# B&R Automation Studio project Genmot_Markalama_ (part 4)

#### GZ1Ax.c - Implementation code
```c
/*******************************************************************
 * COPYRIGHT -- Bernecker + Rainer
 ********************************************************************
 * PROGRAM: Basic
 * File: Basic.c
 * Author: Bernecker + Rainer
 * Created: December 01, 2009
 ********************************************************************
 * Implementation of Program Basic
 ********************************************************************/

#ifdef _DEFAULT_INCLUDES
#include <AsDefault.h>
#endif
#include <string.h>

/* defines of the state-constants */
#define STATE_WAIT              0
#define STATE_POWER_ON          1
#define STATE_HOME              2

#define STATE_READY             10
#define STATE_HALT              11
#define STATE_STOP              12
#define STATE_JOG_POSITIVE      13
#define STATE_JOG_NEGATIVE      14
#define STATE_MOVE_ABSOLUTE     15
#define STATE_MOVE_ADDITIVE     16
#define STATE_MOVE_VELOCITY     17

#define STATE_ERROR_AXIS        100
#define STATE_ERROR             101
#define STATE_ERROR_RESET       102
#define STATE_READ              103

_LOCAL REAL   data;

_INIT void GZ1Axis_init(void)
{

	/* get axis object */
	Axis1Obj = (UDINT)&GZ1_Axis;

	AxisStep = STATE_WAIT;  /* start step */

	GZ1Axis.Parameter.Velocity              = 10000;  /*velocity for movement*/
	GZ1Axis.Parameter.Acceleration          = 10000;  /*acceleration for movement*/
	GZ1Axis.Parameter.Deceleration          = 10000;  /*deceleration for movement*/
	GZ1Axis.Parameter.JogVelocity           = 5000;   /*velocity for jogging */

}

_CYCLIC void GZ1Axis_cyclic(void)
{
	if(GZ1Axis.Command.Power)
	{
		GZ1Axis.Speed.VelocityOverride			= 0.5;
	}

/***************************************************************
        Control Sequence
***************************************************************/

/* status information is read before the step sequencer to attain a shorter reaction time */
/************************ MC_READSTATUS *************************/
	MC_ReadStatus_0.Enable = !MC_ReadStatus_0.Error;
	MC_ReadStatus_0.Axis = Axis1Obj;
	MC_ReadStatus(&MC_ReadStatus_0);
	GZ1Axis.AxisState.Disabled             = MC_ReadStatus_0.Disabled;
	GZ1Axis.AxisState.StandStill           = MC_ReadStatus_0.StandStill;
	GZ1Axis.AxisState.Stopping             = MC_ReadStatus_0.Stopping;
	GZ1Axis.AxisState.Homing               = MC_ReadStatus_0.Homing;
	GZ1Axis.AxisState.DiscreteMotion       = MC_ReadStatus_0.DiscreteMotion;
	GZ1Axis.AxisState.ContinuousMotion     = MC_ReadStatus_0.ContinuousMotion;
	GZ1Axis.AxisState.SynchronizedMotion   = MC_ReadStatus_0.SynchronizedMotion;
	GZ1Axis.AxisState.ErrorStop            = MC_ReadStatus_0.Errorstop;

	/********************MC_BR_READDRIVESTATUS***********************/
	MC_BR_ReadDriveStatus_0.Enable = !MC_BR_ReadDriveStatus_0.Error;
	MC_BR_ReadDriveStatus_0.Axis = Axis1Obj;
	MC_BR_ReadDriveStatus_0.AdrDriveStatus = (UDINT)&(GZ1Axis.Status.DriveStatus);
	MC_BR_ReadDriveStatus(&MC_BR_ReadDriveStatus_0);

	/******************** MC_READACTUALPOSITION *********************/
	MC_ReadActualPosition_0.Enable = (!MC_ReadActualPosition_0.Error);
	MC_ReadActualPosition_0.Axis = Axis1Obj;
	MC_ReadActualPosition(&MC_ReadActualPosition_0);
	if(MC_ReadActualPosition_0.Valid == 1)
	{
		GZ1Axis.Status.ActPosition = MC_ReadActualPosition_0.Position;
	}

	/******************** MC_READACTUALVELOCITY *********************/
	MC_ReadActualVelocity_0.Enable = (!MC_ReadActualVelocity_0.Error);
	MC_ReadActualVelocity_0.Axis = Axis1Obj;
	MC_ReadActualVelocity(&MC_ReadActualVelocity_0);
	if(MC_ReadActualVelocity_0.Valid == 1)
	{
		GZ1Axis.Status.ActVelocity = MC_ReadActualVelocity_0.Velocity;
	}

	/*********************** MC SET OVERRIDE *********************/
	MC_SetOverride_0.Enable = (!MC_SetOverride_0.Error);
	MC_SetOverride_0.AccFactor = GZ1Axis.Speed.AccelerationOverride = 1.0;
	if ((GZ1Axis.Speed.VelocityOverride < 2.01) && (GZ1Axis.Speed.VelocityOverride > 0.0000001))
	{
		MC_SetOverride_0.VelFactor = GZ1Axis.Speed.VelocityOverride;
	}
	MC_SetOverride_0.Axis=Axis1Obj;
	MC_SetOverride(&MC_SetOverride_0);

	/************************ MC_READAXISERROR **********************/
	MC_ReadAxisError_0.Enable = !MC_ReadAxisError_0.Error;
	MC_ReadAxisError_0.Axis = Axis1Obj;
	MC_ReadAxisError_0.DataAddress = (UDINT)&(GZ1Axis.Status.ErrorText);
	MC_ReadAxisError_0.DataLength = sizeof(GZ1Axis.Status.ErrorText);
	strcpy((void*)&MC_ReadAxisError_0.DataObjectName,"acp10etxen");
	MC_ReadAxisError(&MC_ReadAxisError_0);

	/* central monitoring of stop command attains a shorter reaction time in case of emergency stop */
	/******************CHECK for STOP COMMAND************************/
	if (GZ1Axis.Command.Stop == 1)
	{
		if ((AxisStep >= STATE_READY) && (AxisStep < STATE_ERROR))
		{
			/* reset all FB execute inputs we use */
			MC_Home_0.Execute = 0;
			MC_Stop_0.Execute = 0;
			MC_MoveAbsolute_0.Execute = 0;
			MC_MoveAdditive_0.Execute = 0;
			MC_MoveVelocity_0.Execute = 0;
			MC_ReadAxisError_0.Acknowledge = 0;
			MC_Reset_0.Execute = 0;

			/* reset user commands */
			GZ1Axis.Command.Stop = 0;
			GZ1Axis.Command.Home = 0;
			GZ1Axis.Command.MoveJogPos = 0;
			GZ1Axis.Command.MoveJogNeg = 0;
			GZ1Axis.Command.MoveVelocity = 0;
			GZ1Axis.Command.MoveAbsolute = 0;
			GZ1Axis.Command.MoveAdditive = 0;
			AxisStep = STATE_STOP;
		}
	}

	/**************** CHECK FOR GENERAL AXIS ERROR ******************/
	if ((MC_ReadAxisError_0.AxisErrorID != 0) && (MC_ReadAxisError_0.Valid == 1))
	{
		AxisStep = STATE_ERROR_AXIS;
	}
		/***************** CHECK IF POWER SHOULD BE OFF *******************/
	else if ((GZ1Axis.Command.Power == 0) && (MC_ReadAxisError_0.Valid == 1))
	{
		if ((MC_ReadStatus_0.Errorstop == 1) && (MC_ReadStatus_0.Valid == 1))
		{
			AxisStep = STATE_ERROR_RESET;
		}
		else
		{
			AxisStep = STATE_WAIT;
		}
	}

	switch(AxisStep)
	{
		/******************** WAIT *************************/
		case STATE_WAIT:  /* STATE: Wait */
			if (GZ1Axis.Command.Power == 1)
			{
				AxisStep = STATE_POWER_ON;
			}
			else
			{
				MC_Power_0.Enable = 0;

			}

			/* reset all FB execute inputs we use */
			MC_Home_0.Execute = 0;
			MC_Stop_0.Execute = 0;
			MC_MoveAbsolute_0.Execute = 0;
			MC_MoveAdditive_0.Execute = 0;
			MC_MoveVelocity_0.Execute = 0;
			MC_ReadAxisError_0.Acknowledge = 0;
			MC_Reset_0.Execute = 0;

			/* reset user commands */
			GZ1Axis.Command.Stop = 0;
			GZ1Axis.Command.Home = 0;
			GZ1Axis.Command.MoveJogPos = 0;
			GZ1Axis.Command.MoveJogNeg = 0;
			GZ1Axis.Command.MoveVelocity = 0;
			GZ1Axis.Command.MoveAbsolute = 0;
			GZ1Axis.Command.MoveAdditive = 0;

			GZ1Axis.Status.ErrorID = 0;
			break;

		/******************** POWER ON **********************/
		case STATE_POWER_ON:  /* STATE: Power on */
			MC_Power_0.Enable = 1;
			if (MC_Power_0.Status == 1)
			{
				if (!GZ1HomeOk & Parametreler_0.Z_HomeStart)
				{
					GZ1Axis.Command.Home = 1;
				}
			    AxisStep = STATE_READY;
			}
			/* if a power error occured go to error state */
			if (MC_Power_0.Error == 1)
			{
				GZ1Axis.Status.ErrorID = MC_Power_0.ErrorID;
				AxisStep = STATE_ERROR;
			}
			break;

		/******************** READY **********************/
		case STATE_READY:  /* STATE: Waiting for commands */
			if (GZ1Axis.Command.Home == 1)
			{
				GZ1Axis.Command.Home = 0;
				AxisStep = STATE_HOME;
			}
			else if (GZ1Axis.Command.Stop == 1)
			{
				AxisStep = STATE_STOP;
			}
			else if (GZ1Axis.Command.MoveJogPos == 1)
			{
				AxisStep = STATE_JOG_POSITIVE;
			}
			else if (GZ1Axis.Command.MoveJogNeg == 1)
			{
				AxisStep = STATE_JOG_NEGATIVE;
			}
			else if (GZ1Axis.Command.MoveAbsolute == 1)
			{
				GZ1Axis.Command.MoveAbsolute = 0;
				AxisStep = STATE_MOVE_ABSOLUTE;
			}
			else if (GZ1Axis.Command.MoveAdditive == 1)
			{
				GZ1Axis.Command.MoveAdditive = 0;
				AxisStep = STATE_MOVE_ADDITIVE;
			}
			else if (GZ1Axis.Command.MoveVelocity == 1)
			{
				GZ1Axis.Command.MoveVelocity = 0;
				AxisStep = STATE_MOVE_VELOCITY;
			}
			else if (GZ1Axis.Command.Halt == 1)
			{
				GZ1Axis.Command.Halt = 0;
				AxisStep = STATE_HALT;
			}
			break;

		/******************** HOME **********************/
		case STATE_HOME:  /* STATE: start homing process */
			MC_Home_0.Position = GZ1Axis.Parameter.HomePosition;
			MC_Home_0.HomingMode = GZ1Axis.Parameter.HomeMode;
			MC_Home_0.Execute = 1;
			if (MC_Home_0.Done == 1)
			{

				MC_Home_0.Execute = 0;
				AxisStep = STATE_READ;
			}
			/* if a homing error occured go to error state */
			if (MC_Home_0.Error == 1)
			{
				MC_Home_0.Execute = 0;
				GZ1Axis.Status.ErrorID = MC_Home_0.ErrorID;
				AxisStep = STATE_ERROR;
			}
			break;

		/************************HALT MOVEMENT**************************/
		case STATE_HALT:  /* STATE: Stop the active movement */
			MC_Halt_0.Deceleration = GZ1Axis.Parameter.Deceleration;
			MC_Halt_0.Execute = 1;
			if (MC_Halt_0.Done == 1)
			{
				MC_Halt_0.Execute = 0;
				AxisStep = STATE_READY;
			}
			/*check if error occured */
			if (MC_Halt_0.Error == 1)
			{
				MC_Halt_0.Execute = 0;
				GZ1Axis.Status.ErrorID = MC_Halt_0.ErrorID;
				AxisStep = STATE_ERROR;
			}
			break;

		/*********************** STOP MOVEMENT *************************/
		case STATE_STOP: /* STATE: Stop movement as long as command is set */
			MC_Stop_0.Deceleration = GZ1Axis.Parameter.Deceleration;
			MC_Stop_0.Execute = 1;
			/* if axis is stopped go to ready state */
			if ((MC_Stop_0.Done == 1) && (GZ1Axis.Command.Stop == 0))
			{
				MC_Stop_0.Execute = 0;
				AxisStep = STATE_READY;
			}
			/* check if error occured */
			if (MC_Stop_0.Error == 1)
			{
				GZ1Axis.Status.ErrorID = MC_Stop_0.ErrorID;
				MC_Stop_0.Execute = 0;
				AxisStep = STATE_ERROR;
			}
			break;

		/******************** START JOG MOVEMENT POSITVE **********************/
		case STATE_JOG_POSITIVE:  /* STATE: Start jog movement in positive direction */
			MC_MoveVelocity_0.Velocity      = GZ1Axis.Parameter.JogVelocity;
			MC_MoveVelocity_0.Acceleration  = GZ1Axis.Parameter.Acceleration;
			MC_MoveVelocity_0.Deceleration  = GZ1Axis.Parameter.Deceleration;
			MC_MoveVelocity_0.Direction     = mcPOSITIVE_DIR;
			MC_MoveVelocity_0.Execute = 1;
			/* check if jog movement should be stopped */
			if (GZ1Axis.Command.MoveJogPos == 0)
			{
				MC_MoveVelocity_0.Execute = 0;
				AxisStep = STATE_HALT;
			}
			/* check if error occured */
			if (MC_MoveVelocity_0.Error == 1)
			{
				GZ1Axis.Status.ErrorID = MC_MoveVelocity_0.ErrorID;
				MC_MoveVelocity_0.Execute = 0;
				AxisStep = STATE_ERROR;
			}
			break;

		/******************** START JOG MOVEMENT NEGATIVE **********************/
		case STATE_JOG_NEGATIVE:  /* STATE: Start jog movement in negative direction */
			MC_MoveVelocity_0.Velocity      = GZ1Axis.Parameter.JogVelocity;
			MC_MoveVelocity_0.Acceleration  = GZ1Axis.Parameter.Acceleration;
			MC_MoveVelocity_0.Deceleration  = GZ1Axis.Parameter.Deceleration;
			MC_MoveVelocity_0.Direction     = mcNEGATIVE_DIR;
			MC_MoveVelocity_0.Execute = 1;
			/* check if jog movement should be stopped */
			if (GZ1Axis.Command.MoveJogNeg == 0)
			{
				MC_MoveVelocity_0.Execute = 0;
				AxisStep = STATE_HALT;
			}
			/* check if error occured */
			if (MC_MoveVelocity_0.Error == 1)
			{
				GZ1Axis.Status.ErrorID = MC_MoveVelocity_0.ErrorID;
				MC_MoveVelocity_0.Execute = 0;
				AxisStep = STATE_ERROR;
			}
			break;

		/******************** START ABSOLUTE MOVEMENT **********************/
		case STATE_MOVE_ABSOLUTE:  /* STATE: Start absolute movement */
			MC_MoveAbsolute_0.Position      = GZ1Axis.Parameter.Position;
			MC_MoveAbsolute_0.Velocity      = GZ1Axis.Parameter.Velocity;
			MC_MoveAbsolute_0.Acceleration  = GZ1Axis.Parameter.Acceleration;
			MC_MoveAbsolute_0.Deceleration  = GZ1Axis.Parameter.Deceleration;
			MC_MoveAbsolute_0.Direction     = GZ1Axis.Parameter.Direction;
			MC_MoveAbsolute_0.Execute = 1;
			/* check if commanded position is reached */
			if (GZ1Axis.Command.Halt == 1)
			{
				GZ1Axis.Command.Halt = 0;
				MC_MoveAbsolute_0.Execute = 0;
				AxisStep = STATE_HALT;
			}
			else if (MC_MoveAbsolute_0.Done == 1)
			{
				MC_MoveAbsolute_0.Execute = 0;
				AxisStep = STATE_READY;
			}
			/* check if error occured */
			if (MC_MoveAbsolute_0.Error == 1)
			{
				GZ1Axis.Status.ErrorID = MC_MoveAbsolute_0.ErrorID;
				MC_MoveAbsolute_0.Execute = 0;
				AxisStep = STATE_ERROR;
			}
			break;

		/******************** START ADDITIVE MOVEMENT **********************/
		case STATE_MOVE_ADDITIVE:  /* STATE: Start additive movement */
			MC_MoveAdditive_0.Distance      = GZ1Axis.Parameter.Distance;
			MC_MoveAdditive_0.Velocity      = GZ1Axis.Parameter.Velocity;
			MC_MoveAdditive_0.Acceleration  = GZ1Axis.Parameter.Acceleration;
			MC_MoveAdditive_0.Deceleration  = GZ1Axis.Parameter.Deceleration;
			MC_MoveAdditive_0.Execute = 1;
			/* check if commanded distance is reached */
			if (GZ1Axis.Command.Halt == 1)
			{
				GZ1Axis.Command.Halt = 0;
				MC_MoveAdditive_0.Execute = 0;
				AxisStep = STATE_HALT;
			}
			else if (MC_MoveAdditive_0.Done == 1)
			{
				MC_MoveAdditive_0.Execute = 0;
				AxisStep = STATE_READY;
			}
			/* check if error occured */
			if (MC_MoveAdditive_0.Error == 1)
			{
				GZ1Axis.Status.ErrorID = MC_MoveAdditive_0.ErrorID;
				MC_MoveAdditive_0.Execute = 0;
				AxisStep = STATE_ERROR;
			}
			break;

		/******************** START VELOCITY MOVEMENT **********************/
		case STATE_MOVE_VELOCITY:  /* STATE: Start velocity movement */
			MC_MoveVelocity_0.Velocity      = GZ1Axis.Parameter.Velocity;
			MC_MoveVelocity_0.Acceleration  = GZ1Axis.Parameter.Acceleration;
			MC_MoveVelocity_0.Deceleration  = GZ1Axis.Parameter.Deceleration;
			MC_MoveVelocity_0.Direction     = GZ1Axis.Parameter.Direction;
			MC_MoveVelocity_0.Execute = 1;
			/* check if commanded velocity is reached */
			if (GZ1Axis.Command.Halt == 1)
			{
				GZ1Axis.Command.Halt = 0;
				MC_MoveVelocity_0.Execute = 0;
				AxisStep = STATE_HALT;
			}
			else if (MC_MoveVelocity_0.InVelocity == 1)
			{
				MC_MoveVelocity_0.Execute = 0;
				AxisStep = STATE_READY;
			}
			/* check if error occured */
			if (MC_MoveVelocity_0.Error == 1)
			{
				GZ1Axis.Status.ErrorID = MC_MoveVelocity_0.ErrorID;
				MC_MoveVelocity_0.Execute = 0;
				AxisStep = STATE_ERROR;
			}
			break;

		/******************** FB-ERROR OCCURED *************************/
		case STATE_ERROR:  /* STATE: Error */
			/* check if FB indicates an axis error */
			if (MC_ReadAxisError_0.AxisErrorCount != 0)
			{
				AxisStep = STATE_ERROR_AXIS;
			}
			else
			{
				if (GZ1Axis.Command.ErrorAcknowledge == 1)
				{
					GZ1Axis.Command.ErrorAcknowledge = 0;
					GZ1Axis.Status.ErrorID = 0;
					/* reset axis if it is in axis state ErrorStop */
					if ((MC_ReadStatus_0.Errorstop == 1) && (MC_ReadStatus_0.Valid == 1))
					{
						AxisStep = STATE_ERROR_RESET;
					}
					else
					{
						AxisStep = STATE_WAIT;
					}
				}
			}
			break;

		/******************** AXIS-ERROR OCCURED *************************/
		case STATE_ERROR_AXIS:  /* STATE: Axis Error */
			if (MC_ReadAxisError_0.Valid == 1)
			{
				if (MC_ReadAxisError_0.AxisErrorID != 0)
				{
					GZ1Axis.Status.ErrorID = MC_ReadAxisError_0.AxisErrorID;
				}
				MC_ReadAxisError_0.Acknowledge = 0;
				if (GZ1Axis.Command.ErrorAcknowledge == 1)
				{
					GZ1Axis.Command.ErrorAcknowledge = 0;
					/* acknowledge axis error */
					if (MC_ReadAxisError_0.AxisErrorID != 0)
					{
						MC_ReadAxisError_0.Acknowledge = 1;
					}
				}
				if (MC_ReadAxisError_0.AxisErrorCount == 0)
				{
					GZ1Axis.Status.ErrorID = 0;
					/* reset axis if it is in axis state ErrorStop */
					if ((MC_ReadStatus_0.Errorstop == 1) && (MC_ReadStatus_0.Valid == 1))
					{
						AxisStep = STATE_ERROR_RESET;
					}
					else
					{
						AxisStep = STATE_WAIT;
					}
				}
			}
			break;

		/******************** RESET DONE *************************/
		case STATE_ERROR_RESET:  /* STATE: Wait for reset done */
			MC_Reset_0.Execute = 1;
			/* reset MC_Power.Enable if this FB is in Error*/
			if(MC_Power_0.Error == 1)
			{
				MC_Power_0.Enable = 0;
			}
			if(MC_Reset_0.Done == 1)
			{
				MC_Reset_0.Execute = 0;
				AxisStep = STATE_WAIT;
			}
			else if (MC_Reset_0.Error == 1)
			{
				MC_Reset_0.Execute = 0;
				AxisStep = STATE_ERROR;
			}
			break;

		/******************** SEQUENCE END *************************/

		/**********************STATE_READ************************/
		case STATE_READ:
			MC_BR_CyclicRead_0.Enable=1;
			MC_BR_CyclicRead_0.ParID = 277;
			MC_BR_CyclicRead_0.DataAddress = (UDINT)&data;
			MC_BR_CyclicRead_0.DataType =ncPAR_TYP_REAL;

			if (MC_BR_CyclicRead_0.Valid)
			{
				AxisStep = STATE_READY;
			}
			else if (MC_BR_CyclicRead_0.Error)
			{

				GZ1Axis.Status.ErrorID = MC_BR_CyclicRead_0.ErrorID;
				/*Reset Enable before going to STATE_ERROR*/
				MC_BR_CyclicRead_0.Enable=0;
				AxisStep = STATE_ERROR;
			}
			break;  /*end read*/

	}

/***************************************************************
        Function Block Calls
***************************************************************/

/************************** MC_POWER ****************************/
	MC_Power_0.Axis = Axis1Obj;  /* pointer to axis */
	MC_Power(&MC_Power_0);

	/************************** MC_HOME *****************************/
	MC_Home_0.Axis = Axis1Obj;
	MC_Home(&MC_Home_0);

	/********************** MC_MOVEABSOLUTE *************************/
	MC_MoveAbsolute_0.Axis = Axis1Obj;
	MC_MoveAbsolute(&MC_MoveAbsolute_0);

	/********************** MC_MOVEADDITIVE *************************/
	MC_MoveAdditive_0.Axis = Axis1Obj;
	MC_MoveAdditive(&MC_MoveAdditive_0);

	/********************** MC_MOVEVELOCITY *************************/
	MC_MoveVelocity_0.Axis = Axis1Obj;
	MC_MoveVelocity(&MC_MoveVelocity_0);

	/************************** MC_STOP *****************************/
	MC_Stop_0.Axis = Axis1Obj;
	MC_Stop(&MC_Stop_0);

	/**************************MC_HALT*******************************/
	MC_Halt_0.Axis = Axis1Obj;
	MC_Halt(&MC_Halt_0);

	/************************** MC_RESET ****************************/
	MC_Reset_0.Axis = Axis1Obj;
	MC_Reset(&MC_Reset_0);

	MC_BR_CyclicRead_0.Axis = Axis1Obj;
	MC_BR_CyclicRead(&MC_BR_CyclicRead_0);

}
```

#### GZ1Ax.var - Local variables
```iecst
(********************************************************************
 * COPYRIGHT --
 ********************************************************************
 * Program: Reg2Ax
 * File: Reg2Ax.var
 * Author: Coder
 * Created: June 20, 2013
 ********************************************************************
 * Local variables of program Reg2Ax
 ********************************************************************)
VAR
	Axis1Obj : UDINT; (*axis reference*)
	Axis2Obj : UDINT; (*axis reference*)
	AxisStep : USINT; (*current step in the step sequence*)
	AutData : MC_AUTDATA_TYP := (0); (*configuration of the automat*)
	MC_Power_0 : MC_Power; (*Function Block*)
	MC_Home_0 : MC_Home; (*Function Block*)
	MC_Stop_0 : MC_Stop; (*Function Block*)
	MC_MoveVelocity_0 : MC_MoveVelocity; (*Function Block*)
	MC_MoveAbsolute_0 : MC_MoveAbsolute; (*Function Block*)
	MC_MoveAdditive_0 : MC_MoveAdditive; (*Function Block*)
	MC_BR_InitAutData_0 : MC_BR_InitAutData; (*Function Block*)
	MC_BR_AutControl_0 : MC_BR_AutControl; (*Function Block*)
	MC_ReadAxisError_0 : MC_ReadAxisError; (*Function Block*)
	MC_Reset_0 : MC_Reset; (*Function Block*)
	MC_ReadStatus_0 : MC_ReadStatus; (*Function Block*)
	MC_ReadActualPosition_0 : MC_ReadActualPosition; (*Function Block*)
	MC_ReadActualVelocity_0 : MC_ReadActualVelocity; (*Function Block*)
	MC_BR_ReadDriveStatus_0 : MC_BR_ReadDriveStatus; (*Function Block*)
	MC_Halt_0 : MC_Halt; (*Function Block*)
	MC_BR_DownloadCamProfileObj_0 : MC_BR_DownloadCamProfileObj;
	SlaveFactor : REAL;
	MC_BR_Phasing_0 : MC_BR_Phasing;
	ShiftFactor : REAL;
	MC_GearInPos_0 : MC_GearInPos;
	MC_GearOut_0 : MC_GearOut;
	MC_SetOverride_0 : MC_SetOverride;
	MC_BR_CyclicRead_0 : MC_BR_CyclicRead;
END_VAR
```

### Program Logical/RC1AxisControl (ANSIC)

#### GC1Ax.c - Implementation code
```c
/*******************************************************************
 * COPYRIGHT -- Bernecker + Rainer
 ********************************************************************
 * PROGRAM: Basic
 * File: Basic.c
 * Author: Bernecker + Rainer
 * Created: December 01, 2009
 ********************************************************************
 * Implementation of Program Basic
 ********************************************************************/

#ifdef _DEFAULT_INCLUDES
#include <AsDefault.h>
#endif
#include <string.h>

/* defines of the state-constants */
#define STATE_WAIT              0
#define STATE_POWER_ON          1
#define STATE_HOME              2

#define STATE_READY             10
#define STATE_HALT              11
#define STATE_STOP              12
#define STATE_JOG_POSITIVE      13
#define STATE_JOG_NEGATIVE      14
#define STATE_MOVE_ABSOLUTE     15
#define STATE_MOVE_ADDITIVE     16
#define STATE_MOVE_VELOCITY     17

#define STATE_ERROR_AXIS        100
#define STATE_ERROR             101
#define STATE_ERROR_RESET       102
#define STATE_READ              103

_LOCAL REAL   data;

_INIT void GC1Axis_init(void)
{

	/* get axis object */
	Axis1Obj = (UDINT)&GC1_Axis;

	AxisStep = STATE_WAIT;  /* start step */

	GC1Axis.Parameter.Velocity              = 2000;  /*velocity for movement*/
	GC1Axis.Parameter.Acceleration          = 10000;  /*acceleration for movement*/
	GC1Axis.Parameter.Deceleration          = 10000;  /*deceleration for movement*/
	GC1Axis.Parameter.JogVelocity           = 2000;   /*velocity for jogging */

}

_CYCLIC void GC1Axis_cyclic(void)
{
	if(GC1Axis.Command.Power)
	{
		GC1Axis.Speed.VelocityOverride			= 0.5;
	}

/***************************************************************
        Control Sequence
***************************************************************/

/* status information is read before the step sequencer to attain a shorter reaction time */
/************************ MC_READSTATUS *************************/
	MC_ReadStatus_0.Enable = !MC_ReadStatus_0.Error;
	MC_ReadStatus_0.Axis = Axis1Obj;
	MC_ReadStatus(&MC_ReadStatus_0);
	GC1Axis.AxisState.Disabled             = MC_ReadStatus_0.Disabled;
	GC1Axis.AxisState.StandStill           = MC_ReadStatus_0.StandStill;
	GC1Axis.AxisState.Stopping             = MC_ReadStatus_0.Stopping;
	GC1Axis.AxisState.Homing               = MC_ReadStatus_0.Homing;
	GC1Axis.AxisState.DiscreteMotion       = MC_ReadStatus_0.DiscreteMotion;
	GC1Axis.AxisState.ContinuousMotion     = MC_ReadStatus_0.ContinuousMotion;
	GC1Axis.AxisState.SynchronizedMotion   = MC_ReadStatus_0.SynchronizedMotion;
	GC1Axis.AxisState.ErrorStop            = MC_ReadStatus_0.Errorstop;

	/********************MC_BR_READDRIVESTATUS***********************/
	MC_BR_ReadDriveStatus_0.Enable = !MC_BR_ReadDriveStatus_0.Error;
	MC_BR_ReadDriveStatus_0.Axis = Axis1Obj;
	MC_BR_ReadDriveStatus_0.AdrDriveStatus = (UDINT)&(GC1Axis.Status.DriveStatus);
	MC_BR_ReadDriveStatus(&MC_BR_ReadDriveStatus_0);

	/******************** MC_READACTUALPOSITION *********************/
	MC_ReadActualPosition_0.Enable = (!MC_ReadActualPosition_0.Error);
	MC_ReadActualPosition_0.Axis = Axis1Obj;
	MC_ReadActualPosition(&MC_ReadActualPosition_0);
	if(MC_ReadActualPosition_0.Valid == 1)
	{
		GC1Axis.Status.ActPosition = MC_ReadActualPosition_0.Position;
	}

	/******************** MC_READACTUALVELOCITY *********************/
	MC_ReadActualVelocity_0.Enable = (!MC_ReadActualVelocity_0.Error);
	MC_ReadActualVelocity_0.Axis = Axis1Obj;
	MC_ReadActualVelocity(&MC_ReadActualVelocity_0);
	if(MC_ReadActualVelocity_0.Valid == 1)
	{
		GC1Axis.Status.ActVelocity = MC_ReadActualVelocity_0.Velocity;
	}

	/*********************** MC SET OVERRIDE *********************/
	MC_SetOverride_0.Enable = (!MC_SetOverride_0.Error);
	MC_SetOverride_0.AccFactor = GC1Axis.Speed.AccelerationOverride = 1.0;
	if ((GC1Axis.Speed.VelocityOverride < 2.01) && (GC1Axis.Speed.VelocityOverride > 0.0000001))
	{
		MC_SetOverride_0.VelFactor = GC1Axis.Speed.VelocityOverride;
	}
	MC_SetOverride_0.Axis=Axis1Obj;
	MC_SetOverride(&MC_SetOverride_0);

	/************************ MC_READAXISERROR **********************/
	MC_ReadAxisError_0.Enable = !MC_ReadAxisError_0.Error;
	MC_ReadAxisError_0.Axis = Axis1Obj;
	MC_ReadAxisError_0.DataAddress = (UDINT)&(GC1Axis.Status.ErrorText);
	MC_ReadAxisError_0.DataLength = sizeof(GC1Axis.Status.ErrorText);
	strcpy((void*)&MC_ReadAxisError_0.DataObjectName,"acp10etxen");
	MC_ReadAxisError(&MC_ReadAxisError_0);

	/* central monitoring of stop command attains a shorter reaction time in case of emergency stop */
	/******************CHECK for STOP COMMAND************************/
	if (GC1Axis.Command.Stop == 1)
	{
		if ((AxisStep >= STATE_READY) && (AxisStep < STATE_ERROR))
		{
			/* reset all FB execute inputs we use */
			MC_Home_0.Execute = 0;
			MC_Stop_0.Execute = 0;
			MC_MoveAbsolute_0.Execute = 0;
			MC_MoveAdditive_0.Execute = 0;
			MC_MoveVelocity_0.Execute = 0;
			MC_ReadAxisError_0.Acknowledge = 0;
			MC_Reset_0.Execute = 0;

			/* reset user commands */
			GC1Axis.Command.Stop = 0;
			GC1Axis.Command.Home = 0;
			GC1Axis.Command.MoveJogPos = 0;
			GC1Axis.Command.MoveJogNeg = 0;
			GC1Axis.Command.MoveVelocity = 0;
			GC1Axis.Command.MoveAbsolute = 0;
			GC1Axis.Command.MoveAdditive = 0;
			AxisStep = STATE_STOP;
		}
	}

	/**************** CHECK FOR GENERAL AXIS ERROR ******************/
	if ((MC_ReadAxisError_0.AxisErrorID != 0) && (MC_ReadAxisError_0.Valid == 1))
	{
		AxisStep = STATE_ERROR_AXIS;
	}
		/***************** CHECK IF POWER SHOULD BE OFF *******************/
	else if ((GC1Axis.Command.Power == 0) && (MC_ReadAxisError_0.Valid == 1))
	{
		if ((MC_ReadStatus_0.Errorstop == 1) && (MC_ReadStatus_0.Valid == 1))
		{
			AxisStep = STATE_ERROR_RESET;
		}
		else
		{
			AxisStep = STATE_WAIT;
		}
	}

	switch(AxisStep)
	{
		/******************** WAIT *************************/
		case STATE_WAIT:  /* STATE: Wait */
			if (GC1Axis.Command.Power == 1)
			{
				AxisStep = STATE_POWER_ON;
			}
			else
			{
				MC_Power_0.Enable = 0;

			}

			/* reset all FB execute inputs we use */
			MC_Home_0.Execute = 0;
			MC_Stop_0.Execute = 0;
			MC_MoveAbsolute_0.Execute = 0;
			MC_MoveAdditive_0.Execute = 0;
			MC_MoveVelocity_0.Execute = 0;
			MC_ReadAxisError_0.Acknowledge = 0;
			MC_Reset_0.Execute = 0;

			/* reset user commands */
			GC1Axis.Command.Stop = 0;
			GC1Axis.Command.Home = 0;
			GC1Axis.Command.MoveJogPos = 0;
			GC1Axis.Command.MoveJogNeg = 0;
			GC1Axis.Command.MoveVelocity = 0;
			GC1Axis.Command.MoveAbsolute = 0;
			GC1Axis.Command.MoveAdditive = 0;

			GC1Axis.Status.ErrorID = 0;
			break;

		/******************** POWER ON **********************/
		case STATE_POWER_ON:  /* STATE: Power on */
			MC_Power_0.Enable = 1;
			if (MC_Power_0.Status == 1)
			{
				if (Parametreler_0.GC1_HomeStart)
				{
					GC1Axis.Command.Home = 1;
				}
			    AxisStep = STATE_READY;
			}
			/* if a power error occured go to error state */
			if (MC_Power_0.Error == 1)
			{
				GC1Axis.Status.ErrorID = MC_Power_0.ErrorID;
				AxisStep = STATE_ERROR;
			}
			break;

		/******************** READY **********************/
		case STATE_READY:  /* STATE: Waiting for commands */
			if (GC1Axis.Command.Home == 1)
			{
				GC1Axis.Command.Home = 0;
				AxisStep = STATE_HOME;
			}
			else if (GC1Axis.Command.Stop == 1)
			{
				AxisStep = STATE_STOP;
			}
			else if (GC1Axis.Command.MoveJogPos == 1)
			{
				AxisStep = STATE_JOG_POSITIVE;
			}
			else if (GC1Axis.Command.MoveJogNeg == 1)
			{
				AxisStep = STATE_JOG_NEGATIVE;
			}
			else if (GC1Axis.Command.MoveAbsolute == 1)
			{
				GC1Axis.Command.MoveAbsolute = 0;
				AxisStep = STATE_MOVE_ABSOLUTE;
			}
			else if (GC1Axis.Command.MoveAdditive == 1)
			{
				GC1Axis.Command.MoveAdditive = 0;
				AxisStep = STATE_MOVE_ADDITIVE;
			}
			else if (GC1Axis.Command.MoveVelocity == 1)
			{
				GC1Axis.Command.MoveVelocity = 0;
				AxisStep = STATE_MOVE_VELOCITY;
			}
			else if (GC1Axis.Command.Halt == 1)
			{
				GC1Axis.Command.Halt = 0;
				AxisStep = STATE_HALT;
			}
			break;

		/******************** HOME **********************/
		case STATE_HOME:  /* STATE: start homing process */
			if (!GC2Axis.AxisState.SynchronizedMotion)
			{
				MC_Home_0.Position = GC1Axis.Parameter.HomePosition;
				MC_Home_0.HomingMode = GC1Axis.Parameter.HomeMode;
				MC_Home_0.Execute = 1;
				if (MC_Home_0.Done == 1 )
				{
					//

					MC_Home_0.Execute = 0;
					AxisStep = STATE_READ;
				}
				/* if a homing error occured go to error state */
				if (MC_Home_0.Error == 1)
				{
					MC_Home_0.Execute = 0;
					GC1Axis.Status.ErrorID = MC_Home_0.ErrorID;
					AxisStep = STATE_ERROR;
				}
			}
			else
			{
				AxisStep = STATE_READ;
				GC2Axis.Command.GearOut = 1;
				GC2Axis.Command.GearInPos = 0;

			}
			break;

		/************************HALT MOVEMENT**************************/
		case STATE_HALT:  /* STATE: Stop the active movement */
			MC_Halt_0.Deceleration = GC1Axis.Parameter.Deceleration;
			MC_Halt_0.Execute = 1;
			if (MC_Halt_0.Done == 1)
			{
				MC_Halt_0.Execute = 0;
				AxisStep = STATE_READY;
			}
			/*check if error occured */
			if (MC_Halt_0.Error == 1)
			{
				MC_Halt_0.Execute = 0;
				GC1Axis.Status.ErrorID = MC_Halt_0.ErrorID;
				AxisStep = STATE_ERROR;
			}
			break;

		/*********************** STOP MOVEMENT *************************/
		case STATE_STOP: /* STATE: Stop movement as long as command is set */
			MC_Stop_0.Deceleration = GC1Axis.Parameter.Deceleration;
			MC_Stop_0.Execute = 1;
			/* if axis is stopped go to ready state */
			if ((MC_Stop_0.Done == 1) && (GC1Axis.Command.Stop == 0))
			{
				MC_Stop_0.Execute = 0;
				AxisStep = STATE_READY;
			}
			/* check if error occured */
			if (MC_Stop_0.Error == 1)
			{
				GC1Axis.Status.ErrorID = MC_Stop_0.ErrorID;
				MC_Stop_0.Execute = 0;
				AxisStep = STATE_ERROR;
			}
			break;

		/******************** START JOG MOVEMENT POSITVE **********************/
		case STATE_JOG_POSITIVE:  /* STATE: Start jog movement in positive direction */
			MC_MoveVelocity_0.Velocity      = GC1Axis.Parameter.JogVelocity;
			MC_MoveVelocity_0.Acceleration  = GC1Axis.Parameter.Acceleration;
			MC_MoveVelocity_0.Deceleration  = GC1Axis.Parameter.Deceleration;
			MC_MoveVelocity_0.Direction     = mcPOSITIVE_DIR;
			MC_MoveVelocity_0.Execute = 1;
			/* check if jog movement should be stopped */
			if (GC1Axis.Command.MoveJogPos == 0)
			{
				MC_MoveVelocity_0.Execute = 0;
				AxisStep = STATE_HALT;
			}
			/* check if error occured */
			if (MC_MoveVelocity_0.Error == 1)
			{
				GC1Axis.Status.ErrorID = MC_MoveVelocity_0.ErrorID;
				MC_MoveVelocity_0.Execute = 0;
				AxisStep = STATE_ERROR;
			}
			break;

		/******************** START JOG MOVEMENT NEGATIVE **********************/
		case STATE_JOG_NEGATIVE:  /* STATE: Start jog movement in negative direction */
			MC_MoveVelocity_0.Velocity      = GC1Axis.Parameter.JogVelocity;
			MC_MoveVelocity_0.Acceleration  = GC1Axis.Parameter.Acceleration;
			MC_MoveVelocity_0.Deceleration  = GC1Axis.Parameter.Deceleration;
			MC_MoveVelocity_0.Direction     = mcNEGATIVE_DIR;
			MC_MoveVelocity_0.Execute = 1;
			/* check if jog movement should be stopped */
			if (GC1Axis.Command.MoveJogNeg == 0)
			{
				MC_MoveVelocity_0.Execute = 0;
				AxisStep = STATE_HALT;
			}
			/* check if error occured */
			if (MC_MoveVelocity_0.Error == 1)
			{
				GC1Axis.Status.ErrorID = MC_MoveVelocity_0.ErrorID;
				MC_MoveVelocity_0.Execute = 0;
				AxisStep = STATE_ERROR;
			}
			break;

		/******************** START ABSOLUTE MOVEMENT **********************/
		case STATE_MOVE_ABSOLUTE:  /* STATE: Start absolute movement */
			MC_MoveAbsolute_0.Position      = GC1Axis.Parameter.Position;
			MC_MoveAbsolute_0.Velocity      = GC1Axis.Parameter.Velocity;
			MC_MoveAbsolute_0.Acceleration  = GC1Axis.Parameter.Acceleration;
			MC_MoveAbsolute_0.Deceleration  = GC1Axis.Parameter.Deceleration;
			MC_MoveAbsolute_0.Direction     = GC1Axis.Parameter.Direction;
			MC_MoveAbsolute_0.Execute = 1;
			/* check if commanded position is reached */
			if (GC1Axis.Command.Halt == 1)
			{
				GC1Axis.Command.Halt = 0;
				MC_MoveAbsolute_0.Execute = 0;
				AxisStep = STATE_HALT;
			}
			else if (MC_MoveAbsolute_0.Done == 1)
			{
				MC_MoveAbsolute_0.Execute = 0;
				AxisStep = STATE_READY;
			}
			/* check if error occured */
			if (MC_MoveAbsolute_0.Error == 1)
			{
				GC1Axis.Status.ErrorID = MC_MoveAbsolute_0.ErrorID;
				MC_MoveAbsolute_0.Execute = 0;
				AxisStep = STATE_ERROR;
			}
			break;

		/******************** START ADDITIVE MOVEMENT **********************/
		case STATE_MOVE_ADDITIVE:  /* STATE: Start additive movement */
			MC_MoveAdditive_0.Distance      = GC1Axis.Parameter.Distance;
			MC_MoveAdditive_0.Velocity      = GC1Axis.Parameter.Velocity;
			MC_MoveAdditive_0.Acceleration  = GC1Axis.Parameter.Acceleration;
			MC_MoveAdditive_0.Deceleration  = GC1Axis.Parameter.Deceleration;
			MC_MoveAdditive_0.Execute = 1;
			/* check if commanded distance is reached */
			if (GC1Axis.Command.Halt == 1)
			{
				GC1Axis.Command.Halt = 0;
				MC_MoveAdditive_0.Execute = 0;
				AxisStep = STATE_HALT;
			}
			else if (MC_MoveAdditive_0.Done == 1)
			{
				MC_MoveAdditive_0.Execute = 0;
				AxisStep = STATE_READY;
			}
			/* check if error occured */
			if (MC_MoveAdditive_0.Error == 1)
			{
				GC1Axis.Status.ErrorID = MC_MoveAdditive_0.ErrorID;
				MC_MoveAdditive_0.Execute = 0;
				AxisStep = STATE_ERROR;
			}
			break;

		/******************** START VELOCITY MOVEMENT **********************/
		case STATE_MOVE_VELOCITY:  /* STATE: Start velocity movement */
			MC_MoveVelocity_0.Velocity      = GC1Axis.Parameter.Velocity;
			MC_MoveVelocity_0.Acceleration  = GC1Axis.Parameter.Acceleration;
			MC_MoveVelocity_0.Deceleration  = GC1Axis.Parameter.Deceleration;
			MC_MoveVelocity_0.Direction     = GC1Axis.Parameter.Direction;
			MC_MoveVelocity_0.Execute = 1;
			/* check if commanded velocity is reached */
			if (GC1Axis.Command.Halt == 1)
			{
				GC1Axis.Command.Halt = 0;
				MC_MoveVelocity_0.Execute = 0;
				AxisStep = STATE_HALT;
			}
			else if (MC_MoveVelocity_0.InVelocity == 1)
			{
				MC_MoveVelocity_0.Execute = 0;
				AxisStep = STATE_READY;
			}
			/* check if error occured */
			if (MC_MoveVelocity_0.Error == 1)
			{
				GC1Axis.Status.ErrorID = MC_MoveVelocity_0.ErrorID;
				MC_MoveVelocity_0.Execute = 0;
				AxisStep = STATE_ERROR;
			}
			break;

		/******************** FB-ERROR OCCURED *************************/
		case STATE_ERROR:  /* STATE: Error */
			/* check if FB indicates an axis error */
			if (MC_ReadAxisError_0.AxisErrorCount != 0)
			{
				AxisStep = STATE_ERROR_AXIS;
			}
			else
			{
				if (GC1Axis.Command.ErrorAcknowledge == 1)
				{
					GC1Axis.Command.ErrorAcknowledge = 0;
					GC1Axis.Status.ErrorID = 0;
					/* reset axis if it is in axis state ErrorStop */
					if ((MC_ReadStatus_0.Errorstop == 1) && (MC_ReadStatus_0.Valid == 1))
					{
						AxisStep = STATE_ERROR_RESET;
					}
					else
					{
						AxisStep = STATE_WAIT;
					}
				}
			}
			break;

		/******************** AXIS-ERROR OCCURED *************************/
		case STATE_ERROR_AXIS:  /* STATE: Axis Error */
			if (MC_ReadAxisError_0.Valid == 1)
			{
				if (MC_ReadAxisError_0.AxisErrorID != 0)
				{
					GC1Axis.Status.ErrorID = MC_ReadAxisError_0.AxisErrorID;
				}
				MC_ReadAxisError_0.Acknowledge = 0;
				if (GC1Axis.Command.ErrorAcknowledge == 1)
				{
					GC1Axis.Command.ErrorAcknowledge = 0;
					/* acknowledge axis error */
					if (MC_ReadAxisError_0.AxisErrorID != 0)
					{
						MC_ReadAxisError_0.Acknowledge = 1;
					}
				}
				if (MC_ReadAxisError_0.AxisErrorCount == 0)
				{
					GC1Axis.Status.ErrorID = 0;
					/* reset axis if it is in axis state ErrorStop */
					if ((MC_ReadStatus_0.Errorstop == 1) && (MC_ReadStatus_0.Valid == 1))
					{
						AxisStep = STATE_ERROR_RESET;
					}
					else
					{
						AxisStep = STATE_WAIT;
					}
				}
			}
			break;

		/******************** RESET DONE *************************/
		case STATE_ERROR_RESET:  /* STATE: Wait for reset done */
			MC_Reset_0.Execute = 1;
			/* reset MC_Power.Enable if this FB is in Error*/
			if(MC_Power_0.Error == 1)
			{
				MC_Power_0.Enable = 0;
			}
			if(MC_Reset_0.Done == 1)
			{
				MC_Reset_0.Execute = 0;
				AxisStep = STATE_WAIT;
			}
			else if (MC_Reset_0.Error == 1)
			{
				MC_Reset_0.Execute = 0;
				AxisStep = STATE_ERROR;
			}
			break;

		/******************** SEQUENCE END *************************/

		/**********************STATE_READ************************/
		case STATE_READ:
			MC_BR_CyclicRead_0.Enable=1;
			MC_BR_CyclicRead_0.ParID = 277;
			MC_BR_CyclicRead_0.DataAddress = (UDINT)&data;
			MC_BR_CyclicRead_0.DataType =ncPAR_TYP_REAL;

			if (MC_BR_CyclicRead_0.Valid)
			{
				AxisStep = STATE_READY;
			}
			else if (MC_BR_CyclicRead_0.Error)
			{

				GC1Axis.Status.ErrorID = MC_BR_CyclicRead_0.ErrorID;
				/*Reset Enable before going to STATE_ERROR*/
				MC_BR_CyclicRead_0.Enable=0;
				AxisStep = STATE_ERROR;
			}
			break;  /*end read*/

	}

/***************************************************************
        Function Block Calls
***************************************************************/

/************************** MC_POWER ****************************/
	MC_Power_0.Axis = Axis1Obj;  /* pointer to axis */
	MC_Power(&MC_Power_0);

	/************************** MC_HOME *****************************/
	MC_Home_0.Axis = Axis1Obj;
	MC_Home(&MC_Home_0);

	/********************** MC_MOVEABSOLUTE *************************/
	MC_MoveAbsolute_0.Axis = Axis1Obj;
	MC_MoveAbsolute(&MC_MoveAbsolute_0);

	/********************** MC_MOVEADDITIVE *************************/
	MC_MoveAdditive_0.Axis = Axis1Obj;
	MC_MoveAdditive(&MC_MoveAdditive_0);

	/********************** MC_MOVEVELOCITY *************************/
	MC_MoveVelocity_0.Axis = Axis1Obj;
	MC_MoveVelocity(&MC_MoveVelocity_0);

	/************************** MC_STOP *****************************/
	MC_Stop_0.Axis = Axis1Obj;
	MC_Stop(&MC_Stop_0);

	/**************************MC_HALT*******************************/
	MC_Halt_0.Axis = Axis1Obj;
	MC_Halt(&MC_Halt_0);

	/************************** MC_RESET ****************************/
	MC_Reset_0.Axis = Axis1Obj;
	MC_Reset(&MC_Reset_0);

	MC_BR_CyclicRead_0.Axis = Axis1Obj;
	MC_BR_CyclicRead(&MC_BR_CyclicRead_0);

}
```

### Program Logical/RC2AxisControl (ANSIC)

#### GC2Ax.c - Implementation code
```c
/*******************************************************************
 * COPYRIGHT -- Bernecker + Rainer
 ********************************************************************
 * PROGRAM: Basic
 * File: Basic.c
 * Author: Bernecker + Rainer
 * Created: December 01, 2009
 ********************************************************************
 * Implementation of Program Basic
 ********************************************************************/

#ifdef _DEFAULT_INCLUDES
#include <AsDefault.h>
#endif
#include <string.h>

/* defines of the state-constants */
#define STATE_WAIT              0
#define STATE_POWER_ON          1
#define STATE_HOME              2

#define STATE_READY             10
#define STATE_HALT              11
#define STATE_STOP              12
#define STATE_JOG_POSITIVE      13
#define STATE_JOG_NEGATIVE      14
#define STATE_MOVE_ABSOLUTE     15
#define STATE_MOVE_ADDITIVE     16
#define STATE_MOVE_VELOCITY     17
#define STATE_GEAR_IN           40
#define STATE_GEAR_OUT          50

#define STATE_ERROR_AXIS        100
#define STATE_ERROR             101
#define STATE_ERROR_RESET       102
#define STATE_READ              103

_LOCAL REAL   data;

_INIT void GC2Axis_init(void)
{

	/* get axis object */
	Axis1Obj = (UDINT)&GC1_Axis;
    Axis2Obj = (UDINT)&GC2_Axis;

	AxisStep = STATE_WAIT;  /* start step */

	GC2Axis.Parameter.Velocity              = 2000;  /*velocity for movement*/
	GC2Axis.Parameter.Acceleration          = 10000;  /*acceleration for movement*/
	GC2Axis.Parameter.Deceleration          = 10000;  /*deceleration for movement*/
	GC2Axis.Parameter.JogVelocity           = 2000;   /*velocity for jogging */

}

_CYCLIC void GC2Axis_cyclic(void)
{
	if(GC2Axis.Command.Power)
	{
		GC2Axis.Speed.VelocityOverride			= 0.5;
	}

/***************************************************************
        Control Sequence
***************************************************************/

/* status information is read before the step sequencer to attain a shorter reaction time */
/************************ MC_READSTATUS *************************/
	MC_ReadStatus_0.Enable = !MC_ReadStatus_0.Error;
	MC_ReadStatus_0.Axis = Axis2Obj;
	MC_ReadStatus(&MC_ReadStatus_0);
	GC2Axis.AxisState.Disabled             = MC_ReadStatus_0.Disabled;
	GC2Axis.AxisState.StandStill           = MC_ReadStatus_0.StandStill;
	GC2Axis.AxisState.Stopping             = MC_ReadStatus_0.Stopping;
	GC2Axis.AxisState.Homing               = MC_ReadStatus_0.Homing;
	GC2Axis.AxisState.DiscreteMotion       = MC_ReadStatus_0.DiscreteMotion;
	GC2Axis.AxisState.ContinuousMotion     = MC_ReadStatus_0.ContinuousMotion;
	GC2Axis.AxisState.SynchronizedMotion   = MC_ReadStatus_0.SynchronizedMotion;
	GC2Axis.AxisState.ErrorStop            = MC_ReadStatus_0.Errorstop;

	/********************MC_BR_READDRIVESTATUS***********************/
	MC_BR_ReadDriveStatus_0.Enable = !MC_BR_ReadDriveStatus_0.Error;
	MC_BR_ReadDriveStatus_0.Axis = Axis2Obj;
	MC_BR_ReadDriveStatus_0.AdrDriveStatus = (UDINT)&(GC2Axis.Status.DriveStatus);
	MC_BR_ReadDriveStatus(&MC_BR_ReadDriveStatus_0);

	/******************** MC_READACTUALPOSITION *********************/
	MC_ReadActualPosition_0.Enable = (!MC_ReadActualPosition_0.Error);
	MC_ReadActualPosition_0.Axis = Axis2Obj;
	MC_ReadActualPosition(&MC_ReadActualPosition_0);
	if(MC_ReadActualPosition_0.Valid == 1)
	{
		GC2Axis.Status.ActPosition = MC_ReadActualPosition_0.Position;
	}

	/******************** MC_READACTUALVELOCITY *********************/
	MC_ReadActualVelocity_0.Enable = (!MC_ReadActualVelocity_0.Error);
	MC_ReadActualVelocity_0.Axis = Axis2Obj;
	MC_ReadActualVelocity(&MC_ReadActualVelocity_0);
	if(MC_ReadActualVelocity_0.Valid == 1)
	{
		GC2Axis.Status.ActVelocity = MC_ReadActualVelocity_0.Velocity;
	}

	/*********************** MC SET OVERRIDE *********************/
	MC_SetOverride_0.Enable = (!MC_SetOverride_0.Error);
	MC_SetOverride_0.AccFactor = GC2Axis.Speed.AccelerationOverride = 1.0;
	if ((GC2Axis.Speed.VelocityOverride < 2.01) && (GC2Axis.Speed.VelocityOverride > 0.0000001))
	{
		MC_SetOverride_0.VelFactor = GC2Axis.Speed.VelocityOverride;
	}
	MC_SetOverride_0.Axis=Axis2Obj;
	MC_SetOverride(&MC_SetOverride_0);

	/************************ MC_READAXISERROR **********************/
	MC_ReadAxisError_0.Enable = !MC_ReadAxisError_0.Error;
	MC_ReadAxisError_0.Axis = Axis2Obj;
	MC_ReadAxisError_0.DataAddress = (UDINT)&(GC2Axis.Status.ErrorText);
	MC_ReadAxisError_0.DataLength = sizeof(GC2Axis.Status.ErrorText);
	strcpy((void*)&MC_ReadAxisError_0.DataObjectName,"acp10etxen");
	MC_ReadAxisError(&MC_ReadAxisError_0);

	/* central monitoring of stop command attains a shorter reaction time in case of emergency stop */
	/******************CHECK for STOP COMMAND************************/
	if (GC2Axis.Command.Stop == 1)
	{
		if ((AxisStep >= STATE_READY) && (AxisStep < STATE_ERROR))
		{
			/* reset all FB execute inputs we use */
			MC_Home_0.Execute = 0;
			MC_Stop_0.Execute = 0;
			MC_MoveAbsolute_0.Execute = 0;
			MC_MoveAdditive_0.Execute = 0;
			MC_MoveVelocity_0.Execute = 0;
			MC_ReadAxisError_0.Acknowledge = 0;
			MC_Reset_0.Execute = 0;

			/* reset user commands */
			GC2Axis.Command.Stop = 0;
			GC2Axis.Command.Home = 0;
			GC2Axis.Command.MoveJogPos = 0;
			GC2Axis.Command.MoveJogNeg = 0;
			GC2Axis.Command.MoveVelocity = 0;
			GC2Axis.Command.MoveAbsolute = 0;
			GC2Axis.Command.MoveAdditive = 0;
			AxisStep = STATE_STOP;
		}
	}

	/**************** CHECK FOR GENERAL AXIS ERROR ******************/
	if ((MC_ReadAxisError_0.AxisErrorID != 0) && (MC_ReadAxisError_0.Valid == 1))
	{
		AxisStep = STATE_ERROR_AXIS;
	}
		/***************** CHECK IF POWER SHOULD BE OFF *******************/
	else if ((GC2Axis.Command.Power == 0) && (MC_ReadAxisError_0.Valid == 1))
	{
		if ((MC_ReadStatus_0.Errorstop == 1) && (MC_ReadStatus_0.Valid == 1))
		{
			AxisStep = STATE_ERROR_RESET;
		}
		else
		{
			AxisStep = STATE_WAIT;
		}
	}

	switch(AxisStep)
	{
		/******************** WAIT *************************/
		case STATE_WAIT:  /* STATE: Wait */
			if (GC2Axis.Command.Power == 1)
			{
				AxisStep = STATE_POWER_ON;
			}
			else
			{
				MC_Power_0.Enable = 0;

			}

			/* reset all FB execute inputs we use */
			MC_Home_0.Execute = 0;
			MC_Stop_0.Execute = 0;
			MC_MoveAbsolute_0.Execute = 0;
			MC_MoveAdditive_0.Execute = 0;
			MC_MoveVelocity_0.Execute = 0;
			MC_ReadAxisError_0.Acknowledge = 0;
			MC_Reset_0.Execute = 0;

			/* reset user commands */
			GC2Axis.Command.Stop = 0;
			GC2Axis.Command.Home = 0;
			GC2Axis.Command.MoveJogPos = 0;
			GC2Axis.Command.MoveJogNeg = 0;
			GC2Axis.Command.MoveVelocity = 0;
			GC2Axis.Command.MoveAbsolute = 0;
			GC2Axis.Command.MoveAdditive = 0;

			GC2Axis.Status.ErrorID = 0;
			break;

		/******************** POWER ON **********************/
		case STATE_POWER_ON:  /* STATE: Power on */
			MC_Power_0.Enable = 1;
			if (MC_Power_0.Status == 1)
			{
				if (Parametreler_0.GC2_HomeStart)
				{
					GC2Axis.Command.Home = 1;
				}
			    AxisStep = STATE_READY;
			}
			/* if a power error occured go to error state */
			if (MC_Power_0.Error == 1)
			{
				GC2Axis.Status.ErrorID = MC_Power_0.ErrorID;
				AxisStep = STATE_ERROR;
			}
			break;

		/******************** READY **********************/
		case STATE_READY:  /* STATE: Waiting for commands */
			if (GC2Axis.Command.Home == 1)
			{
				GC2Axis.Command.Home = 0;
				AxisStep = STATE_HOME;
			}
			else if (GC2Axis.Command.Stop == 1)
			{
				AxisStep = STATE_STOP;
			}
			else if (GC2Axis.Command.MoveJogPos == 1)
			{
				AxisStep = STATE_JOG_POSITIVE;
			}
			else if (GC2Axis.Command.MoveJogNeg == 1)
			{
				AxisStep = STATE_JOG_NEGATIVE;
			}
			else if (GC2Axis.Command.MoveAbsolute == 1)
			{
				GC2Axis.Command.MoveAbsolute = 0;
				AxisStep = STATE_MOVE_ABSOLUTE;
			}
			else if (GC2Axis.Command.MoveAdditive == 1)
			{
				GC2Axis.Command.MoveAdditive = 0;
				AxisStep = STATE_MOVE_ADDITIVE;
			}
			else if (GC2Axis.Command.MoveVelocity == 1)
			{
				GC2Axis.Command.MoveVelocity = 0;
				AxisStep = STATE_MOVE_VELOCITY;
			}
			else if (GC2Axis.Command.GearInPos == 1)
			{
				GC2Axis.Command.GearInPos = 0;
				AxisStep = STATE_GEAR_IN;
			}
			else if (GC2Axis.Command.GearOut == 1)
			{
				GC2Axis.Command.GearOut = 0;
				AxisStep = STATE_GEAR_OUT;
			}
			else if (GC2Axis.Command.Halt == 1)
			{
				GC2Axis.Command.Halt = 0;
				AxisStep = STATE_HALT;
			}
			break;

		/******************** HOME **********************/
		case STATE_HOME:  /* STATE: start homing process */
			if (!GC2Axis.AxisState.SynchronizedMotion)
			{
				MC_Home_0.Position = GC2Axis.Parameter.HomePosition;
				MC_Home_0.HomingMode = GC2Axis.Parameter.HomeMode;
				MC_Home_0.Execute = 1;
				if (MC_Home_0.Done == 1)
				{

					MC_Home_0.Execute = 0;
					AxisStep = STATE_READ;

				}
				/* if a homing error occured go to error state */
				if (MC_Home_0.Error == 1)
				{
					MC_Home_0.Execute = 0;
					GC2Axis.Status.ErrorID = MC_Home_0.ErrorID;
					AxisStep = STATE_ERROR;
				}
			}
			else
			{

				AxisStep = STATE_READ;
				GC2Axis.Command.GearInPos = 0;
				GC2Axis.Command.GearOut = 1;

			}
			break;

		/************************HALT MOVEMENT**************************/
		case STATE_HALT:  /* STATE: Stop the active movement */
			MC_Halt_0.Deceleration = GC2Axis.Parameter.Deceleration;
			MC_Halt_0.Execute = 1;
			if (MC_Halt_0.Done == 1)
			{
				MC_Halt_0.Execute = 0;
				AxisStep = STATE_READY;
			}
			/*check if error occured */
			if (MC_Halt_0.Error == 1)
			{
				MC_Halt_0.Execute = 0;
				GC2Axis.Status.ErrorID = MC_Halt_0.ErrorID;
				AxisStep = STATE_ERROR;
			}
			break;

		/*********************** STOP MOVEMENT *************************/
		case STATE_STOP: /* STATE: Stop movement as long as command is set */
			MC_Stop_0.Deceleration = GC2Axis.Parameter.Deceleration;
			MC_Stop_0.Execute = 1;
			/* if axis is stopped go to ready state */
			if ((MC_Stop_0.Done == 1) && (GC2Axis.Command.Stop == 0))
			{
				MC_Stop_0.Execute = 0;
				AxisStep = STATE_READY;
			}
			/* check if error occured */
			if (MC_Stop_0.Error == 1)
			{
				GC2Axis.Status.ErrorID = MC_Stop_0.ErrorID;
				MC_Stop_0.Execute = 0;
				AxisStep = STATE_ERROR;
			}
			break;

		/******************** START JOG MOVEMENT POSITVE **********************/
		case STATE_JOG_POSITIVE:  /* STATE: Start jog movement in positive direction */
			MC_MoveVelocity_0.Velocity      = GC2Axis.Parameter.JogVelocity;
			MC_MoveVelocity_0.Acceleration  = GC2Axis.Parameter.Acceleration;
			MC_MoveVelocity_0.Deceleration  = GC2Axis.Parameter.Deceleration;
			MC_MoveVelocity_0.Direction     = mcPOSITIVE_DIR;
			MC_MoveVelocity_0.Execute = 1;
			/* check if jog movement should be stopped */
			if (GC2Axis.Command.MoveJogPos == 0)
			{
				MC_MoveVelocity_0.Execute = 0;
				AxisStep = STATE_HALT;
			}
			/* check if error occured */
			if (MC_MoveVelocity_0.Error == 1)
			{
				GC2Axis.Status.ErrorID = MC_MoveVelocity_0.ErrorID;
				MC_MoveVelocity_0.Execute = 0;
				AxisStep = STATE_ERROR;
			}
			break;

		/******************** START JOG MOVEMENT NEGATIVE **********************/
		case STATE_JOG_NEGATIVE:  /* STATE: Start jog movement in negative direction */
			MC_MoveVelocity_0.Velocity      = GC2Axis.Parameter.JogVelocity;
			MC_MoveVelocity_0.Acceleration  = GC2Axis.Parameter.Acceleration;
			MC_MoveVelocity_0.Deceleration  = GC2Axis.Parameter.Deceleration;
			MC_MoveVelocity_0.Direction     = mcNEGATIVE_DIR;
			MC_MoveVelocity_0.Execute = 1;
			/* check if jog movement should be stopped */
			if (GC2Axis.Command.MoveJogNeg == 0)
			{
				MC_MoveVelocity_0.Execute = 0;
				AxisStep = STATE_HALT;
			}
			/* check if error occured */
			if (MC_MoveVelocity_0.Error == 1)
			{
				GC2Axis.Status.ErrorID = MC_MoveVelocity_0.ErrorID;
				MC_MoveVelocity_0.Execute = 0;
				AxisStep = STATE_ERROR;
			}
			break;

		/******************** START ABSOLUTE MOVEMENT **********************/
		case STATE_MOVE_ABSOLUTE:  /* STATE: Start absolute movement */
			MC_MoveAbsolute_0.Position      = GC2Axis.Parameter.Position;
			MC_MoveAbsolute_0.Velocity      = GC2Axis.Parameter.Velocity;
			MC_MoveAbsolute_0.Acceleration  = GC2Axis.Parameter.Acceleration;
			MC_MoveAbsolute_0.Deceleration  = GC2Axis.Parameter.Deceleration;
			MC_MoveAbsolute_0.Direction     = GC2Axis.Parameter.Direction;
			MC_MoveAbsolute_0.Execute = 1;
			/* check if commanded position is reached */
			if (GC2Axis.Command.Halt == 1)
			{
				GC2Axis.Command.Halt = 0;
				MC_MoveAbsolute_0.Execute = 0;
				AxisStep = STATE_HALT;
			}
			else if (MC_MoveAbsolute_0.Done == 1)
			{
				MC_MoveAbsolute_0.Execute = 0;
				AxisStep = STATE_READY;
			}
			/* check if error occured */
			if (MC_MoveAbsolute_0.Error == 1)
			{
				GC2Axis.Status.ErrorID = MC_MoveAbsolute_0.ErrorID;
				MC_MoveAbsolute_0.Execute = 0;
				AxisStep = STATE_ERROR;
			}
			break;

		/******************** START ADDITIVE MOVEMENT **********************/
		case STATE_MOVE_ADDITIVE:  /* STATE: Start additive movement */
			MC_MoveAdditive_0.Distance      = GC2Axis.Parameter.Distance;
			MC_MoveAdditive_0.Velocity      = GC2Axis.Parameter.Velocity;
			MC_MoveAdditive_0.Acceleration  = GC2Axis.Parameter.Acceleration;
			MC_MoveAdditive_0.Deceleration  = GC2Axis.Parameter.Deceleration;
			MC_MoveAdditive_0.Execute = 1;
			/* check if commanded distance is reached */
			if (GC2Axis.Command.Halt == 1)
			{
				GC2Axis.Command.Halt = 0;
				MC_MoveAdditive_0.Execute = 0;
				AxisStep = STATE_HALT;
			}
			else if (MC_MoveAdditive_0.Done == 1)
			{
				MC_MoveAdditive_0.Execute = 0;
				AxisStep = STATE_READY;
			}
			/* check if error occured */
			if (MC_MoveAdditive_0.Error == 1)
			{
				GC2Axis.Status.ErrorID = MC_MoveAdditive_0.ErrorID;
				MC_MoveAdditive_0.Execute = 0;
				AxisStep = STATE_ERROR;
			}
			break;

		/******************** START VELOCITY MOVEMENT **********************/
		case STATE_MOVE_VELOCITY:  /* STATE: Start velocity movement */
			MC_MoveVelocity_0.Velocity      = GC2Axis.Parameter.Velocity;
			MC_MoveVelocity_0.Acceleration  = GC2Axis.Parameter.Acceleration;
			MC_MoveVelocity_0.Deceleration  = GC2Axis.Parameter.Deceleration;
			MC_MoveVelocity_0.Direction     = GC2Axis.Parameter.Direction;
			MC_MoveVelocity_0.Execute = 1;
			/* check if commanded velocity is reached */
			if (GC2Axis.Command.Halt == 1)
			{
				GC2Axis.Command.Halt = 0;
				MC_MoveVelocity_0.Execute = 0;
				AxisStep = STATE_HALT;
			}
			else if (MC_MoveVelocity_0.InVelocity == 1)
			{
				MC_MoveVelocity_0.Execute = 0;
				AxisStep = STATE_READY;
			}
			/* check if error occured */
			if (MC_MoveVelocity_0.Error == 1)
			{
				GC2Axis.Status.ErrorID = MC_MoveVelocity_0.ErrorID;
				MC_MoveVelocity_0.Execute = 0;
				AxisStep = STATE_ERROR;
			}
			break;

		case STATE_GEAR_IN:  /* engage slave and master with set gear ratio*/
			MC_GearIn_0.RatioNumerator=1000;  /*1:2 Slave/Master ratio*/
			MC_GearIn_0.RatioDenominator=1000;  /*1:2 Slave/Master ratio*/
			MC_GearIn_0.Acceleration=50000;
			MC_GearIn_0.Deceleration=50000;
			MC_GearIn_0.Execute=1;
			/*Return to wait state once slave is in gear*/
			if (MC_GearIn_0.InGear)
			{
				MC_GearIn_0.Execute=0;
				AxisStep=STATE_READY;
			}
			else if (MC_GearIn_0.Error)
			{
				GC2Axis.Status.ErrorID=MC_GearIn_0.ErrorID;
				MC_GearIn_0.Execute=0;
				AxisStep=STATE_ERROR;
			}
			break;

		/******************** GEAR OUT*************************/
		case STATE_GEAR_OUT:
			MC_GearOut_0.Execute=1;
			/*Return to wait state once gear out is complete*/
			if (MC_GearOut_0.Done)
			{
				MC_GearOut_0.Execute=0;
				AxisStep = STATE_READY;
			}
			else if (MC_GearOut_0.Error)
			{
				GC2Axis.Status.ErrorID = MC_GearOut_0.ErrorID;
				MC_GearOut_0.Execute=0;
				AxisStep = STATE_ERROR;
			}
			break;

		/******************** FB-ERROR OCCURED *************************/
		case STATE_ERROR:  /* STATE: Error */
			/* check if FB indicates an axis error */
			if (MC_ReadAxisError_0.AxisErrorCount != 0)
			{
				AxisStep = STATE_ERROR_AXIS;
			}
			else
			{
				if (GC2Axis.Command.ErrorAcknowledge == 1)
				{
					GC2Axis.Command.ErrorAcknowledge = 0;
					GC2Axis.Status.ErrorID = 0;
					/* reset axis if it is in axis state ErrorStop */
					if ((MC_ReadStatus_0.Errorstop == 1) && (MC_ReadStatus_0.Valid == 1))
					{
						AxisStep = STATE_ERROR_RESET;
					}
					else
					{
						AxisStep = STATE_WAIT;
					}
				}
			}
			break;

		/******************** AXIS-ERROR OCCURED *************************/
		case STATE_ERROR_AXIS:  /* STATE: Axis Error */
			if (MC_ReadAxisError_0.Valid == 1)
			{
				if (MC_ReadAxisError_0.AxisErrorID != 0)
				{
					GC2Axis.Status.ErrorID = MC_ReadAxisError_0.AxisErrorID;
				}
				MC_ReadAxisError_0.Acknowledge = 0;
				if (GC2Axis.Command.ErrorAcknowledge == 1)
				{
					GC2Axis.Command.ErrorAcknowledge = 0;
					/* acknowledge axis error */
					if (MC_ReadAxisError_0.AxisErrorID != 0)
					{
						MC_ReadAxisError_0.Acknowledge = 1;
					}
				}
				if (MC_ReadAxisError_0.AxisErrorCount == 0)
				{
					GC2Axis.Status.ErrorID = 0;
					/* reset axis if it is in axis state ErrorStop */
					if ((MC_ReadStatus_0.Errorstop == 1) && (MC_ReadStatus_0.Valid == 1))
					{
						AxisStep = STATE_ERROR_RESET;
					}
					else
					{
						AxisStep = STATE_WAIT;
					}
				}
			}
			break;

		/******************** RESET DONE *************************/
		case STATE_ERROR_RESET:  /* STATE: Wait for reset done */
			MC_Reset_0.Execute = 1;
			/* reset MC_Power.Enable if this FB is in Error*/
			if(MC_Power_0.Error == 1)
			{
				MC_Power_0.Enable = 0;
			}
			if(MC_Reset_0.Done == 1)
			{
				MC_Reset_0.Execute = 0;
				AxisStep = STATE_WAIT;
			}
			else if (MC_Reset_0.Error == 1)
			{
				MC_Reset_0.Execute = 0;
				AxisStep = STATE_ERROR;
			}
			break;

		/******************** SEQUENCE END *************************/

		/**********************STATE_READ************************/
		case STATE_READ:
			MC_BR_CyclicRead_0.Enable=1;
			MC_BR_CyclicRead_0.ParID = 277;
			MC_BR_CyclicRead_0.DataAddress = (UDINT)&data;
			MC_BR_CyclicRead_0.DataType =ncPAR_TYP_REAL;

			if (MC_BR_CyclicRead_0.Valid)
			{
				AxisStep = STATE_READY;
			}
			else if (MC_BR_CyclicRead_0.Error)
			{

				GC2Axis.Status.ErrorID = MC_BR_CyclicRead_0.ErrorID;
				/*Reset Enable before going to STATE_ERROR*/
				MC_BR_CyclicRead_0.Enable=0;
				AxisStep = STATE_ERROR;
			}
			break;  /*end read*/

	}

/***************************************************************
        Function Block Calls
***************************************************************/

/************************** MC_POWER ****************************/
	MC_Power_0.Axis = Axis2Obj;  /* pointer to axis */
	MC_Power(&MC_Power_0);

	/************************** MC_HOME *****************************/
	MC_Home_0.Axis = Axis2Obj;
	MC_Home(&MC_Home_0);

	/********************** MC_MOVEABSOLUTE *************************/
	MC_MoveAbsolute_0.Axis = Axis2Obj;
	MC_MoveAbsolute(&MC_MoveAbsolute_0);

	/********************** MC_MOVEADDITIVE *************************/
	MC_MoveAdditive_0.Axis = Axis2Obj;
	MC_MoveAdditive(&MC_MoveAdditive_0);

	/********************** MC_MOVEVELOCITY *************************/
	MC_MoveVelocity_0.Axis = Axis2Obj;
	MC_MoveVelocity(&MC_MoveVelocity_0);

	/************************** MC_STOP *****************************/
	MC_Stop_0.Axis = Axis2Obj;
	MC_Stop(&MC_Stop_0);

	/**************************MC_HALT*******************************/
	MC_Halt_0.Axis = Axis2Obj;
	MC_Halt(&MC_Halt_0);

	/************************** MC_RESET ****************************/
	MC_Reset_0.Axis = Axis2Obj;
	MC_Reset(&MC_Reset_0);

	MC_BR_CyclicRead_0.Axis = Axis2Obj;
	MC_BR_CyclicRead(&MC_BR_CyclicRead_0);

	/************************** MC_GEARIN ***************************/
	MC_GearIn_0.Master=Axis1Obj;  /*Master(virtual) axis*/
	MC_GearIn_0.Slave=Axis2Obj;  /*Slave(real) axis*/
	MC_GearIn(&MC_GearIn_0);

	/************************** MC_GEAROUT **************************/
	MC_GearOut_0.Slave=Axis2Obj;  /*Slave(real) axis*/
	MC_GearOut(&MC_GearOut_0);

}
```

#### GC2Ax.var - Local variables
```iecst
(********************************************************************
 * COPYRIGHT --
 ********************************************************************
 * Program: Reg2Ax
 * File: Reg2Ax.var
 * Author: Coder
 * Created: June 20, 2013
 ********************************************************************
 * Local variables of program Reg2Ax
 ********************************************************************)
VAR
	Axis1Obj : UDINT; (*axis reference*)
	Axis2Obj : UDINT; (*axis reference*)
	AxisStep : USINT; (*current step in the step sequence*)
	AutData : MC_AUTDATA_TYP := (0); (*configuration of the automat*)
	MC_Power_0 : MC_Power; (*Function Block*)
	MC_Home_0 : MC_Home; (*Function Block*)
	MC_Stop_0 : MC_Stop; (*Function Block*)
	MC_MoveVelocity_0 : MC_MoveVelocity; (*Function Block*)
	MC_MoveAbsolute_0 : MC_MoveAbsolute; (*Function Block*)
	MC_MoveAdditive_0 : MC_MoveAdditive; (*Function Block*)
	MC_BR_InitAutData_0 : MC_BR_InitAutData; (*Function Block*)
	MC_BR_AutControl_0 : MC_BR_AutControl; (*Function Block*)
	MC_ReadAxisError_0 : MC_ReadAxisError; (*Function Block*)
	MC_Reset_0 : MC_Reset; (*Function Block*)
	MC_ReadStatus_0 : MC_ReadStatus; (*Function Block*)
	MC_ReadActualPosition_0 : MC_ReadActualPosition; (*Function Block*)
	MC_ReadActualVelocity_0 : MC_ReadActualVelocity; (*Function Block*)
	MC_BR_ReadDriveStatus_0 : MC_BR_ReadDriveStatus; (*Function Block*)
	MC_Halt_0 : MC_Halt; (*Function Block*)
	MC_BR_DownloadCamProfileObj_0 : MC_BR_DownloadCamProfileObj;
	SlaveFactor : REAL;
	MC_BR_Phasing_0 : MC_BR_Phasing;
	ShiftFactor : REAL;
	MC_GearIn_0 : MC_GearIn;
	MC_GearOut_0 : MC_GearOut;
	MC_SetOverride_0 : MC_SetOverride;
	MC_BR_CyclicRead_0 : MC_BR_CyclicRead;
END_VAR
```

### Program Logical/GRXAxisControl (ANSIC)

#### GRXAx.c - Implementation code
```c
/*******************************************************************
 * COPYRIGHT -- Bernecker + Rainer
 ********************************************************************
 * PROGRAM: Basic
 * File: Basic.c
 * Author: Bernecker + Rainer
 * Created: December 01, 2009
 ********************************************************************
 * Implementation of Program Basic
 ********************************************************************/

#ifdef _DEFAULT_INCLUDES
#include <AsDefault.h>
#endif
#include <string.h>

/* defines of the state-constants */
#define STATE_WAIT              0
#define STATE_POWER_ON          1
#define STATE_HOME              2

#define STATE_READY             10
#define STATE_HALT              11
#define STATE_STOP              12
#define STATE_JOG_POSITIVE      13
#define STATE_JOG_NEGATIVE      14
#define STATE_MOVE_ABSOLUTE     15
#define STATE_MOVE_ADDITIVE     16
#define STATE_MOVE_VELOCITY     17

#define STATE_ERROR_AXIS        100
#define STATE_ERROR             101
#define STATE_ERROR_RESET       102
#define STATE_READ              103

_LOCAL REAL   data;

_INIT void GRXAxis_init(void)
{

	/* get axis object */
	Axis1Obj = (UDINT)&GRX_Axis;

	AxisStep = STATE_WAIT;  /* start step */

	GRXAxis.Parameter.Velocity              = 50000;  /*velocity for movement*/
	GRXAxis.Parameter.Acceleration          = 80000;  /*acceleration for movement*/
	GRXAxis.Parameter.Deceleration          = 80000;  /*deceleration for movement*/
	GRXAxis.Parameter.JogVelocity           = 20000;   /*velocity for jogging */
	GRXAxis.Speed.VelocityOverride			= 1.0;

}

_CYCLIC void GRXAxis_cyclic(void)
{
//	if(GRXAxis.Command.Power)
//	{
//	GRXAxis.Speed.VelocityOverride			= 1.0;
//	}

/***************************************************************
        Control Sequence
***************************************************************/

/* status information is read before the step sequencer to attain a shorter reaction time */
/************************ MC_READSTATUS *************************/
	MC_ReadStatus_0.Enable = !MC_ReadStatus_0.Error;
	MC_ReadStatus_0.Axis = Axis1Obj;
	MC_ReadStatus(&MC_ReadStatus_0);
	GRXAxis.AxisState.Disabled             = MC_ReadStatus_0.Disabled;
	GRXAxis.AxisState.StandStill           = MC_ReadStatus_0.StandStill;
	GRXAxis.AxisState.Stopping             = MC_ReadStatus_0.Stopping;
	GRXAxis.AxisState.Homing               = MC_ReadStatus_0.Homing;
	GRXAxis.AxisState.DiscreteMotion       = MC_ReadStatus_0.DiscreteMotion;
	GRXAxis.AxisState.ContinuousMotion     = MC_ReadStatus_0.ContinuousMotion;
	GRXAxis.AxisState.SynchronizedMotion   = MC_ReadStatus_0.SynchronizedMotion;
	GRXAxis.AxisState.ErrorStop            = MC_ReadStatus_0.Errorstop;

	/********************MC_BR_READDRIVESTATUS***********************/
	MC_BR_ReadDriveStatus_0.Enable = !MC_BR_ReadDriveStatus_0.Error;
	MC_BR_ReadDriveStatus_0.Axis = Axis1Obj;
	MC_BR_ReadDriveStatus_0.AdrDriveStatus = (UDINT)&(GRXAxis.Status.DriveStatus);
	MC_BR_ReadDriveStatus(&MC_BR_ReadDriveStatus_0);

	/******************** MC_READACTUALPOSITION *********************/
	MC_ReadActualPosition_0.Enable = (!MC_ReadActualPosition_0.Error);
	MC_ReadActualPosition_0.Axis = Axis1Obj;
	MC_ReadActualPosition(&MC_ReadActualPosition_0);
	if(MC_ReadActualPosition_0.Valid == 1)
	{
		GRXAxis.Status.ActPosition = MC_ReadActualPosition_0.Position;
	}

	/******************** MC_READACTUALVELOCITY *********************/
	MC_ReadActualVelocity_0.Enable = (!MC_ReadActualVelocity_0.Error);
	MC_ReadActualVelocity_0.Axis = Axis1Obj;
	MC_ReadActualVelocity(&MC_ReadActualVelocity_0);
	if(MC_ReadActualVelocity_0.Valid == 1)
	{
		GRXAxis.Status.ActVelocity = MC_ReadActualVelocity_0.Velocity;
	}

	/*********************** MC SET OVERRIDE *********************/
	MC_SetOverride_0.Enable = (!MC_SetOverride_0.Error);
	MC_SetOverride_0.AccFactor = GRXAxis.Speed.AccelerationOverride = 1.0;
	if ((GRXAxis.Speed.VelocityOverride < 2.01) && (GRXAxis.Speed.VelocityOverride > 0.0000001))
	{
		MC_SetOverride_0.VelFactor = GRXAxis.Speed.VelocityOverride;
	}
	MC_SetOverride_0.Axis=Axis1Obj;
	MC_SetOverride(&MC_SetOverride_0);

	/************************ MC_READAXISERROR **********************/
	MC_ReadAxisError_0.Enable = !MC_ReadAxisError_0.Error;
	MC_ReadAxisError_0.Axis = Axis1Obj;
	MC_ReadAxisError_0.DataAddress = (UDINT)&(GRXAxis.Status.ErrorText);
	MC_ReadAxisError_0.DataLength = sizeof(GRXAxis.Status.ErrorText);
	strcpy((void*)&MC_ReadAxisError_0.DataObjectName,"acp10etxen");
	MC_ReadAxisError(&MC_ReadAxisError_0);

	/* central monitoring of stop command attains a shorter reaction time in case of emergency stop */
	/******************CHECK for STOP COMMAND************************/
	if (GRXAxis.Command.Stop == 1)
	{
		if ((AxisStep >= STATE_READY) && (AxisStep < STATE_ERROR))
		{
			/* reset all FB execute inputs we use */
			MC_Home_0.Execute = 0;
			MC_Stop_0.Execute = 0;
			MC_MoveAbsolute_0.Execute = 0;
			MC_MoveAdditive_0.Execute = 0;
			MC_MoveVelocity_0.Execute = 0;
			MC_ReadAxisError_0.Acknowledge = 0;
			MC_Reset_0.Execute = 0;

			/* reset user commands */
			GRXAxis.Command.Stop = 0;
			GRXAxis.Command.Home = 0;
			GRXAxis.Command.MoveJogPos = 0;
			GRXAxis.Command.MoveJogNeg = 0;
			GRXAxis.Command.MoveVelocity = 0;
			GRXAxis.Command.MoveAbsolute = 0;
			GRXAxis.Command.MoveAdditive = 0;
			AxisStep = STATE_STOP;
		}
	}

	/**************** CHECK FOR GENERAL AXIS ERROR ******************/
	if ((MC_ReadAxisError_0.AxisErrorID != 0) && (MC_ReadAxisError_0.Valid == 1))
	{
		AxisStep = STATE_ERROR_AXIS;
	}
		/***************** CHECK IF POWER SHOULD BE OFF *******************/
	else if ((GRXAxis.Command.Power == 0) && (MC_ReadAxisError_0.Valid == 1))
	{
		if ((MC_ReadStatus_0.Errorstop == 1) && (MC_ReadStatus_0.Valid == 1))
		{
			AxisStep = STATE_ERROR_RESET;
		}
		else
		{
			AxisStep = STATE_WAIT;
		}
	}

	switch(AxisStep)
	{
		/******************** WAIT *************************/
		case STATE_WAIT:  /* STATE: Wait */
			if (GRXAxis.Command.Power == 1)
			{
				AxisStep = STATE_POWER_ON;
			}
			else
			{
				MC_Power_0.Enable = 0;

			}

			/* reset all FB execute inputs we use */
			MC_Home_0.Execute = 0;
			MC_Stop_0.Execute = 0;
			MC_MoveAbsolute_0.Execute = 0;
			MC_MoveAdditive_0.Execute = 0;
			MC_MoveVelocity_0.Execute = 0;
			MC_ReadAxisError_0.Acknowledge = 0;
			MC_Reset_0.Execute = 0;

			/* reset user commands */
			GRXAxis.Command.Stop = 0;
			GRXAxis.Command.Home = 0;
			GRXAxis.Command.MoveJogPos = 0;
			GRXAxis.Command.MoveJogNeg = 0;
			GRXAxis.Command.MoveVelocity = 0;
			GRXAxis.Command.MoveAbsolute = 0;
			GRXAxis.Command.MoveAdditive = 0;

			GRXAxis.Status.ErrorID = 0;
			break;

		/******************** POWER ON **********************/
		case STATE_POWER_ON:  /* STATE: Power on */
			MC_Power_0.Enable = 1;
			if (MC_Power_0.Status == 1)
			{
				if (!GRXHomeOk)
				{
					GRXAxis.Command.Home = 1;
				}
			    AxisStep = STATE_READY;
			}
			/* if a power error occured go to error state */
			if (MC_Power_0.Error == 1)
			{
				GRXAxis.Status.ErrorID = MC_Power_0.ErrorID;
				AxisStep = STATE_ERROR;
			}
			break;

		/******************** READY **********************/
		case STATE_READY:  /* STATE: Waiting for commands */
			if (GRXAxis.Command.Home == 1)
			{
				GRXAxis.Command.Home = 0;
				AxisStep = STATE_HOME;
			}
			else if (GRXAxis.Command.Stop == 1)
			{
				AxisStep = STATE_STOP;
			}
			else if (GRXAxis.Command.MoveJogPos == 1)
			{
				AxisStep = STATE_JOG_POSITIVE;
			}
			else if (GRXAxis.Command.MoveJogNeg == 1)
			{
				AxisStep = STATE_JOG_NEGATIVE;
			}
			else if (GRXAxis.Command.MoveAbsolute == 1)
			{
				GRXAxis.Command.MoveAbsolute = 0;
				AxisStep = STATE_MOVE_ABSOLUTE;
			}
			else if (GRXAxis.Command.MoveAdditive == 1)
			{
				GRXAxis.Command.MoveAdditive = 0;
				AxisStep = STATE_MOVE_ADDITIVE;
			}
			else if (GRXAxis.Command.MoveVelocity == 1)
			{
				GRXAxis.Command.MoveVelocity = 0;
				AxisStep = STATE_MOVE_VELOCITY;
			}
			else if (GRXAxis.Command.Halt == 1)
			{
				GRXAxis.Command.Halt = 0;
				AxisStep = STATE_HALT;
			}
			break;

		/******************** HOME **********************/
		case STATE_HOME:  /* STATE: start homing process */
			MC_Home_0.Position = GRXAxis.Parameter.HomePosition;
			MC_Home_0.HomingMode = GRXAxis.Parameter.HomeMode;
			MC_Home_0.Execute = 1;
			if (MC_Home_0.Done == 1)
			{

				MC_Home_0.Execute = 0;
				AxisStep = STATE_READ;
			}
			/* if a homing error occured go to error state */
			if (MC_Home_0.Error == 1)
			{
				MC_Home_0.Execute = 0;
				GRXAxis.Status.ErrorID = MC_Home_0.ErrorID;
				AxisStep = STATE_ERROR;
			}
			break;

		/************************HALT MOVEMENT**************************/
		case STATE_HALT:  /* STATE: Stop the active movement */
			MC_Halt_0.Deceleration = GRXAxis.Parameter.Deceleration;
			MC_Halt_0.Execute = 1;
			if (MC_Halt_0.Done == 1)
			{
				MC_Halt_0.Execute = 0;
				AxisStep = STATE_READY;
			}
			/*check if error occured */
			if (MC_Halt_0.Error == 1)
			{
				MC_Halt_0.Execute = 0;
				GRXAxis.Status.ErrorID = MC_Halt_0.ErrorID;
				AxisStep = STATE_ERROR;
			}
			break;

		/*********************** STOP MOVEMENT *************************/
		case STATE_STOP: /* STATE: Stop movement as long as command is set */
			MC_Stop_0.Deceleration = GRXAxis.Parameter.Deceleration;
			MC_Stop_0.Execute = 1;
			/* if axis is stopped go to ready state */
			if ((MC_Stop_0.Done == 1) && (GRXAxis.Command.Stop == 0))
			{
				MC_Stop_0.Execute = 0;
				AxisStep = STATE_READY;
			}
			/* check if error occured */
			if (MC_Stop_0.Error == 1)
			{
				GRXAxis.Status.ErrorID = MC_Stop_0.ErrorID;
				MC_Stop_0.Execute = 0;
				AxisStep = STATE_ERROR;
			}
			break;

		/******************** START JOG MOVEMENT POSITVE **********************/
		case STATE_JOG_POSITIVE:  /* STATE: Start jog movement in positive direction */
			MC_MoveVelocity_0.Velocity      = GRXAxis.Parameter.JogVelocity;
			MC_MoveVelocity_0.Acceleration  = GRXAxis.Parameter.Acceleration;
			MC_MoveVelocity_0.Deceleration  = GRXAxis.Parameter.Deceleration;
			MC_MoveVelocity_0.Direction     = mcPOSITIVE_DIR;
			MC_MoveVelocity_0.Execute = 1;
			/* check if jog movement should be stopped */
			if (GRXAxis.Command.MoveJogPos == 0)
			{
				MC_MoveVelocity_0.Execute = 0;
				AxisStep = STATE_HALT;
			}
			/* check if error occured */
			if (MC_MoveVelocity_0.Error == 1)
			{
				GRXAxis.Status.ErrorID = MC_MoveVelocity_0.ErrorID;
				MC_MoveVelocity_0.Execute = 0;
				AxisStep = STATE_ERROR;
			}
			break;

		/******************** START JOG MOVEMENT NEGATIVE **********************/
		case STATE_JOG_NEGATIVE:  /* STATE: Start jog movement in negative direction */
			MC_MoveVelocity_0.Velocity      = GRXAxis.Parameter.JogVelocity;
			MC_MoveVelocity_0.Acceleration  = GRXAxis.Parameter.Acceleration;
			MC_MoveVelocity_0.Deceleration  = GRXAxis.Parameter.Deceleration;
			MC_MoveVelocity_0.Direction     = mcNEGATIVE_DIR;
			MC_MoveVelocity_0.Execute = 1;
			/* check if jog movement should be stopped */
			if (GRXAxis.Command.MoveJogNeg == 0)
			{
				MC_MoveVelocity_0.Execute = 0;
				AxisStep = STATE_HALT;
			}
			/* check if error occured */
			if (MC_MoveVelocity_0.Error == 1)
			{
				GRXAxis.Status.ErrorID = MC_MoveVelocity_0.ErrorID;
				MC_MoveVelocity_0.Execute = 0;
				AxisStep = STATE_ERROR;
			}
			break;

		/******************** START ABSOLUTE MOVEMENT **********************/
		case STATE_MOVE_ABSOLUTE:  /* STATE: Start absolute movement */
			MC_MoveAbsolute_0.Position      = GRXAxis.Parameter.Position;
			MC_MoveAbsolute_0.Velocity      = GRXAxis.Parameter.Velocity;
			MC_MoveAbsolute_0.Acceleration  = GRXAxis.Parameter.Acceleration;
			MC_MoveAbsolute_0.Deceleration  = GRXAxis.Parameter.Deceleration;
			MC_MoveAbsolute_0.Direction     = GRXAxis.Parameter.Direction;
			MC_MoveAbsolute_0.Execute = 1;
			/* check if commanded position is reached */
			if (GRXAxis.Command.Halt == 1)
			{
				GRXAxis.Command.Halt = 0;
				MC_MoveAbsolute_0.Execute = 0;
				AxisStep = STATE_HALT;
			}
			else if (MC_MoveAbsolute_0.Done == 1)
			{
				MC_MoveAbsolute_0.Execute = 0;
				AxisStep = STATE_READY;
			}
			/* check if error occured */
			if (MC_MoveAbsolute_0.Error == 1)
			{
				GRXAxis.Status.ErrorID = MC_MoveAbsolute_0.ErrorID;
				MC_MoveAbsolute_0.Execute = 0;
				AxisStep = STATE_ERROR;
			}
			break;

		/******************** START ADDITIVE MOVEMENT **********************/
		case STATE_MOVE_ADDITIVE:  /* STATE: Start additive movement */
			MC_MoveAdditive_0.Distance      = GRXAxis.Parameter.Distance;
			MC_MoveAdditive_0.Velocity      = GRXAxis.Parameter.Velocity;
			MC_MoveAdditive_0.Acceleration  = GRXAxis.Parameter.Acceleration;
			MC_MoveAdditive_0.Deceleration  = GRXAxis.Parameter.Deceleration;
			MC_MoveAdditive_0.Execute = 1;
			/* check if commanded distance is reached */
			if (GRXAxis.Command.Halt == 1)
			{
				GRXAxis.Command.Halt = 0;
				MC_MoveAdditive_0.Execute = 0;
				AxisStep = STATE_HALT;
			}
			else if (MC_MoveAdditive_0.Done == 1)
			{
				MC_MoveAdditive_0.Execute = 0;
				AxisStep = STATE_READY;
			}
			/* check if error occured */
			if (MC_MoveAdditive_0.Error == 1)
			{
				GRXAxis.Status.ErrorID = MC_MoveAdditive_0.ErrorID;
				MC_MoveAdditive_0.Execute = 0;
				AxisStep = STATE_ERROR;
			}
			break;

		/******************** START VELOCITY MOVEMENT **********************/
		case STATE_MOVE_VELOCITY:  /* STATE: Start velocity movement */
			MC_MoveVelocity_0.Velocity      = GRXAxis.Parameter.Velocity;
			MC_MoveVelocity_0.Acceleration  = GRXAxis.Parameter.Acceleration;
			MC_MoveVelocity_0.Deceleration  = GRXAxis.Parameter.Deceleration;
			MC_MoveVelocity_0.Direction     = GRXAxis.Parameter.Direction;
			MC_MoveVelocity_0.Execute = 1;
			/* check if commanded velocity is reached */
			if (GRXAxis.Command.Halt == 1)
			{
				GRXAxis.Command.Halt = 0;
				MC_MoveVelocity_0.Execute = 0;
				AxisStep = STATE_HALT;
			}
			else if (MC_MoveVelocity_0.InVelocity == 1)
			{
				MC_MoveVelocity_0.Execute = 0;
				AxisStep = STATE_READY;
			}
			/* check if error occured */
			if (MC_MoveVelocity_0.Error == 1)
			{
				GRXAxis.Status.ErrorID = MC_MoveVelocity_0.ErrorID;
				MC_MoveVelocity_0.Execute = 0;
				AxisStep = STATE_ERROR;
			}
			break;

		/******************** FB-ERROR OCCURED *************************/
		case STATE_ERROR:  /* STATE: Error */
			/* check if FB indicates an axis error */
			if (MC_ReadAxisError_0.AxisErrorCount != 0)
			{
				AxisStep = STATE_ERROR_AXIS;
			}
			else
			{
				if (GRXAxis.Command.ErrorAcknowledge == 1)
				{
					GRXAxis.Command.ErrorAcknowledge = 0;
					GRXAxis.Status.ErrorID = 0;
					/* reset axis if it is in axis state ErrorStop */
					if ((MC_ReadStatus_0.Errorstop == 1) && (MC_ReadStatus_0.Valid == 1))
					{
						AxisStep = STATE_ERROR_RESET;
					}
					else
					{
						AxisStep = STATE_WAIT;
					}
				}
			}
			break;

		/******************** AXIS-ERROR OCCURED *************************/
		case STATE_ERROR_AXIS:  /* STATE: Axis Error */
			if (MC_ReadAxisError_0.Valid == 1)
			{
				if (MC_ReadAxisError_0.AxisErrorID != 0)
				{
					GRXAxis.Status.ErrorID = MC_ReadAxisError_0.AxisErrorID;
				}
				MC_ReadAxisError_0.Acknowledge = 0;
				if (GRXAxis.Command.ErrorAcknowledge == 1)
				{
					GRXAxis.Command.ErrorAcknowledge = 0;
					/* acknowledge axis error */
					if (MC_ReadAxisError_0.AxisErrorID != 0)
					{
						MC_ReadAxisError_0.Acknowledge = 1;
					}
				}
				if (MC_ReadAxisError_0.AxisErrorCount == 0)
				{
					GRXAxis.Status.ErrorID = 0;
					/* reset axis if it is in axis state ErrorStop */
					if ((MC_ReadStatus_0.Errorstop == 1) && (MC_ReadStatus_0.Valid == 1))
					{
						AxisStep = STATE_ERROR_RESET;
					}
					else
					{
						AxisStep = STATE_WAIT;
					}
				}
			}
			break;

		/******************** RESET DONE *************************/
		case STATE_ERROR_RESET:  /* STATE: Wait for reset done */
			MC_Reset_0.Execute = 1;
			/* reset MC_Power.Enable if this FB is in Error*/
			if(MC_Power_0.Error == 1)
			{
				MC_Power_0.Enable = 0;
			}
			if(MC_Reset_0.Done == 1)
			{
				MC_Reset_0.Execute = 0;
				AxisStep = STATE_WAIT;
			}
			else if (MC_Reset_0.Error == 1)
			{
				MC_Reset_0.Execute = 0;
				AxisStep = STATE_ERROR;
			}
			break;

		/******************** SEQUENCE END *************************/

		/**********************STATE_READ************************/
		case STATE_READ:
			MC_BR_CyclicRead_0.Enable=1;
			MC_BR_CyclicRead_0.ParID = 277;
			MC_BR_CyclicRead_0.DataAddress = (UDINT)&data;
			MC_BR_CyclicRead_0.DataType =ncPAR_TYP_REAL;

			if (MC_BR_CyclicRead_0.Valid)
			{
				AxisStep = STATE_READY;
			}
			else if (MC_BR_CyclicRead_0.Error)
			{

				GRXAxis.Status.ErrorID = MC_BR_CyclicRead_0.ErrorID;
				/*Reset Enable before going to STATE_ERROR*/
				MC_BR_CyclicRead_0.Enable=0;
				AxisStep = STATE_ERROR;
			}
			break;  /*end read*/

	}

/***************************************************************
        Function Block Calls
***************************************************************/

/************************** MC_POWER ****************************/
	MC_Power_0.Axis = Axis1Obj;  /* pointer to axis */
	MC_Power(&MC_Power_0);

	/************************** MC_HOME *****************************/
	MC_Home_0.Axis = Axis1Obj;
	MC_Home(&MC_Home_0);

	/********************** MC_MOVEABSOLUTE *************************/
	MC_MoveAbsolute_0.Axis = Axis1Obj;
	MC_MoveAbsolute(&MC_MoveAbsolute_0);

	/********************** MC_MOVEADDITIVE *************************/
	MC_MoveAdditive_0.Axis = Axis1Obj;
	MC_MoveAdditive(&MC_MoveAdditive_0);

	/********************** MC_MOVEVELOCITY *************************/
	MC_MoveVelocity_0.Axis = Axis1Obj;
	MC_MoveVelocity(&MC_MoveVelocity_0);

	/************************** MC_STOP *****************************/
	MC_Stop_0.Axis = Axis1Obj;
	MC_Stop(&MC_Stop_0);

	/**************************MC_HALT*******************************/
	MC_Halt_0.Axis = Axis1Obj;
	MC_Halt(&MC_Halt_0);

	/************************** MC_RESET ****************************/
	MC_Reset_0.Axis = Axis1Obj;
	MC_Reset(&MC_Reset_0);

	MC_BR_CyclicRead_0.Axis = Axis1Obj;
	MC_BR_CyclicRead(&MC_BR_CyclicRead_0);

}
```

### Program Logical/GRYAxisControl (ANSIC) - A new program
